{attribute 'Tc2GvlVarNames'}
{attribute 'strict'}
(* Priorità Pick Point *)
TYPE e_Priorita_PickPoint :
(
	Min_PRIORITY	:= 0,	(* Pick Point con priorità Minima *)
	MAX_PRIORITY	:= 1	(* Pick Point con priorità MASSIMA *)
);
END_TYPE

(* stored: Version 1.1.0.1, ProductVersion 3.1.4024.11
   EnumerationTextList e_Priorita_PickPoint: Id {c51f34ca-fc6f-4b01-84fd-8f8271a8ebfb} *)
